// TIA Portal V19 export
TYPE "lexchangetray_typeUnEmn_toConstraintWorkstationFeedback"
// Type: Bool
// stored: Access Published
   STRUCT
      transferEnable : Bool;   // 允许转移
      trayLiftingCylinderWorkPos : Bool;   // 托盘气缸顶升状态
   END_STRUCT;
END_TYPE
